FUNCTION_BLOCK BasicCalcFibonacci (* Basic FB with empty ECC *)
  (* Standard: 61499-2 *)
  (* Version 1.0, 2023-07-26, AK115394 *)
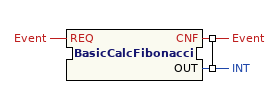
  EVENT_INPUT
    REQ;
  END_EVENT
  EVENT_OUTPUT
    CNF WITH OUT;
  END_EVENT
  VAR_OUTPUT
    OUT : INT;
  END_VAR
  VAR
    Fn0 : INT;
    Fn1 : INT;
    Fnx : INT;
  END_VAR
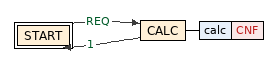
  EC_STATES
    START; (* Initial State *)
    CALC : calc -> CNF;
  END_STATES
  EC_TRANSITIONS
    START TO CALC := REQ;
    CALC TO START := 1;
  END_TRANSITIONS
  ALGORITHM calc IN ST:
VAR_TEMP
	index : SINT;
END_VAR
	Fn0 := 0;
	Fn1 :=1;

    FOR index := 0 TO 20 DO
    	Fnx := Fn0+Fn1;
    	Fn0 := Fn1;
    	Fn1 := Fnx;
    END_FOR;
	OUT:=Fnx;
  END_ALGORITHM
END_FUNCTION_BLOCK
